# EPICS StreamDevice protocol: protocols/caenels.proto
OutTerminator = CR;
InTerminator = CR LF;

getModel {
    out "VER";
    in "#VER:%[^:]:%(\$1)s";
    @init  {
        out "VER";
        in "#VER:%[^:]:%(\$1)s"
    }
}

setEnable {
    out "%{MOFF|MON}";
    in "#AK";
    @mismatch {in "#NAK:%(\$1ErrorMsg-S)d";}
}

setRegulationMode {
    out "LOOP:%{V|I}";
    in "#AK";
    @init {
        out "LOOP:?";
        in "#LOOP:%{V|I}";
    };
}

# the commands are MWV (go to setpt without ramp) and MWVR (ramp)
setVoltage {
    out "MWV%(\$1Rmp-S){|R}:%f";
    in "#AK";
    @mismatch {in "#NAK:%(\$1ErrorMsg-S)d";}
}

# the commands are MWI (go to setpt without ramp) and MWIR (ramp)
setCurrent {
    out "MWI%(\$1Rmp-S){|R}:%f";
    in "#AK";
    @mismatch {in "#NAK:%(\$1ErrorMsg-S)d";}
}

resetStatus {
    out "MRESET";
    in "#AK";
}

getOutputVoltage {
    out "MRV";
    in "#MRV:%f";
}

getOutputCurrent {
    out "MRI";
    in "#MRI:%f";
}

getGroundCurrent {
    out "MGC";
    in "#MGC:%f";
}

getDCLinkVoltage {
    out "MRP";
    in "#MRP:%f";
}

getTemperature {
    out "MRT";
    in "#MRT:%f";
}

getStatusMSB {
    out "MST";
    in "#MST:%4x%*4x";
    @init {
        out "MST";
        in "#MST:%4x%*4x";
    }
}

getStatusLSB {
    out "MST";
    in "#MST:%*4x%4x";
    @init {
        out "MST";
        in "#MST:%*4x%4x";
    }
}

getSlewRateI {
    out "MSRI:?";
    in "#MSRI:%f";
}

getSlewRateV {
    out "MSRV:?";
    in "#MSRV:%f";
}

getOutputPower {
    out "MRW";
    in "#MRW:%f";
}
